// TIA Portal project "HONGPHUONGBAI4TRAM3" (V16)

(* hardware
DEVICE "S7-1200 station_1"  S7-1200 Station
   slot 0: "Rack_0"  S7-1200 Rack  Rack  V1.0
   slot 1: "PLC_1"  CPU 1212C DC/DC/DC  6ES7 212-1AE40-0XB0  V4.3
   slot 2: "DI 16/DQ 16x24VDC_1"  6ES7 223-1BL32-0XB0  V2.0
   slot 3: "DQ 16xRelay_1"  SM 1222 DQ16 x relay  6ES7 222-1HH32-0XB0  V2.0
*)

// ===== PLC "PLC_1"  CPU 1212C DC/DC/DC =====

VAR_GLOBAL   // PLC tag table "Default tag table"
   "STOP" AT %I0.0 : Bool;
   "START" AT %I0.5 : Bool;
   "Tag_3" AT %M0.0 : Bool;
   "A/M" AT %I8.4 : Bool;
   "KM1" AT %Q0.0 : Bool;
   "KM2" AT %Q0.1 : Bool;
   "KM3" AT %Q0.2 : Bool;
   "KM4" AT %Q0.3 : Bool;
   "KM5" AT %Q0.4 : Bool;
   "Tag_1" AT %I0.6 : Bool;
   "Tag_2" AT %I0.7 : Bool;
   "Tag_4" AT %I1.0 : Bool;
   "Tag_5" AT %I1.1 : Bool;
   "Tag_6" AT %I0.1 : Bool;
   "Tag_7" AT %I0.2 : Bool;
   "Tag_8" AT %M0.1 : Bool;
   "Tag_9" AT %M0.2 : Bool;
   "Tag_10" AT %M0.3 : Bool;
   "Tag_11" AT %M0.4 : Bool;
   "Tag_12" AT %M0.5 : Bool;
END_VAR

// folder: System blocks/Program resources

DATA_BLOCK "T1"   // DB1
{ S7_Optimized_Access := 'TRUE' }
AUTHOR : Simatic
FAMILY : IEC
NAME : IEC_TMR
VERSION : 1.0
// stored: InstanceOfName IEC_TIMER
"IEC_TIMER"
BEGIN
END_DATA_BLOCK

// folder: (top level)

ORGANIZATION_BLOCK "Main"   // OB1, LAD, ProgramCycle
TITLE = "Main Program Sweep (Cycle)"
{ S7_Optimized_Access := 'TRUE' }
VERSION : 0.1
   VAR_INPUT
      Initial_Call : Bool;   // Initial call of this OB
      Remanence : Bool;   // =True, if remanent data are available
   END_VAR
BEGIN

REGION Network 1
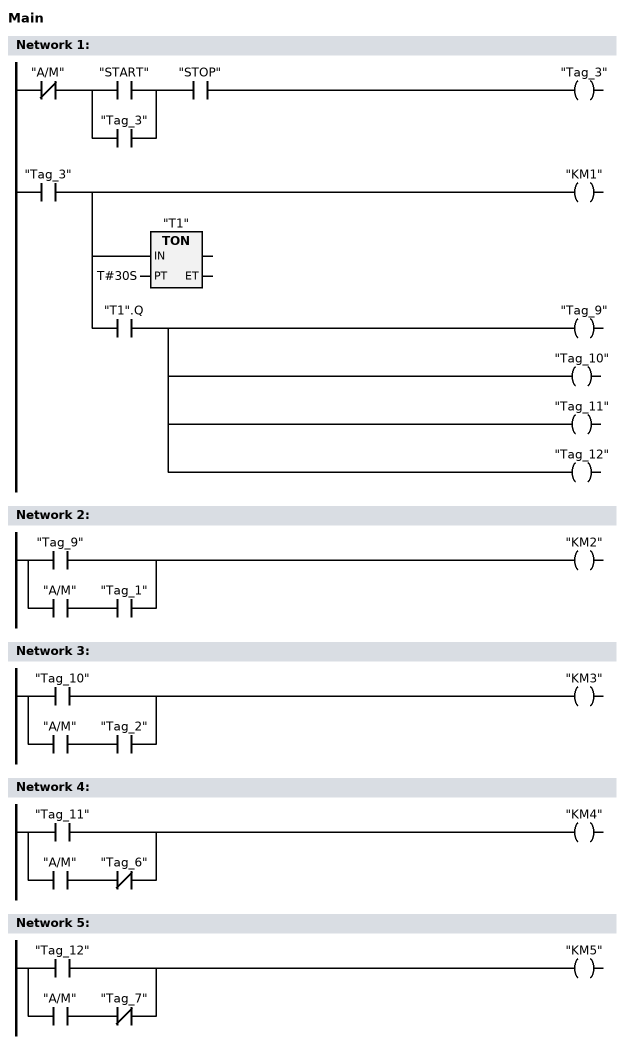
   "Tag_3" := NOT "A/M" AND ("START" OR "Tag_3") AND "STOP";
   "KM1" := "Tag_3";
   "T1".TON(IN := "Tag_3", PT := T#30S);
   "Tag_9" := "Tag_3" AND "T1".Q;
   "Tag_10" := "Tag_9";
   "Tag_11" := "Tag_9";
   "Tag_12" := "Tag_9";
END_REGION

REGION Network 2
   RUNG wire#powerrail
      Contact( "Tag_9" )
      wire#w1
      Coil( "KM2" )
   END_RUNG
   RUNG wire#powerrail
      Contact( "A/M" )
      Contact( "Tag_1" )
   END_RUNG wire#w1
   // the same network as SCL:
   "KM2" := "Tag_9" OR ("A/M" AND "Tag_1");
END_REGION

REGION Network 3
   RUNG wire#powerrail
      Contact( "Tag_10" )
      wire#w1
      Coil( "KM3" )
   END_RUNG
   RUNG wire#powerrail
      Contact( "A/M" )
      Contact( "Tag_2" )
   END_RUNG wire#w1
   // the same network as SCL:
   "KM3" := "Tag_10" OR ("A/M" AND "Tag_2");
END_REGION

REGION Network 4
   RUNG wire#powerrail
      Contact( "Tag_11" )
      wire#w1
      Coil( "KM4" )
   END_RUNG
   RUNG wire#powerrail
      Contact( "A/M" )
      I_Contact( "Tag_6" )
   END_RUNG wire#w1
   // the same network as SCL:
   "KM4" := "Tag_11" OR ("A/M" AND NOT "Tag_6");
END_REGION

REGION Network 5
   RUNG wire#powerrail
      Contact( "Tag_12" )
      wire#w1
      Coil( "KM5" )
   END_RUNG
   RUNG wire#powerrail
      Contact( "A/M" )
      I_Contact( "Tag_7" )
   END_RUNG wire#w1
   // the same network as SCL:
   "KM5" := "Tag_12" OR ("A/M" AND NOT "Tag_7");
END_REGION
END_ORGANIZATION_BLOCK